# EPICS substitutions: Switch.substitutions
file Switch.db
{
pattern {S, TA, DN}
        {BL4A, Keithley, switcher}
}
